# EPICS substitutions: gtsApp/Db/user.substitutions
#device substitutions file

file "db/dbSubExample.db" {
    { user = "numexo2" }
}
